{attribute 'linkalways'} 
{attribute 'no_explicit_call' := 'This FB is a CLASS and must be accessed using methods or properties'}
{attribute 'enable_dynamic_creation'}
FUNCTION_BLOCK FINAL NE_DWORD EXTENDS Node
VAR
	in1 : _DWORD(0);
	in2 : _DWORD(0);
	out : _BOOL(FALSE);
END_VAR

METHOD PUBLIC Clone : I_Node
VAR
	pNode : POINTER TO NE_DWORD;
END_VAR
pNode := __NEW(NE_DWORD);
Clone := pNode^;
END_METHOD

METHOD FB_init : BOOL
VAR_INPUT
	bInitRetains : BOOL; // if TRUE, the retain variables are initialized (warm start / cold start)
	bInCopyCode : BOOL;  // if TRUE, the instance afterwards gets moved into the copy code (online change)
END_VAR
AddInput('in1',THIS^.in1);
AddInput('in2',THIS^.in2);
AddOutput('out', THIS^.out);
END_METHOD

METHOD PROTECTED OnExecute
VAR
END_VAR
out.Value := in1.Value <> in2.Value;
END_METHOD

END_FUNCTION_BLOCK

(* stored: Version 1.1.0.1, ProductVersion 3.1.4024.15
   POU NE_DWORD: Id {d4cfcd26-c402-4334-bbc9-1595d6f2b7ce}, SpecialFunc None
   Folder Constructor: Id {23b6ce0a-7a3f-4e13-97c7-dbc5e52fc27c}
   Method Clone: Id {e3eedafd-cf4d-4c63-9373-ec18b3300aaa}
   Method FB_init: Id {bdb38f08-0be6-42a1-8b0f-328c700b49aa}
   Method OnExecute: Id {6c83cf26-c521-407d-9086-188e5dee254a} *)
